KUKA KRL program: Milling_2_1.src

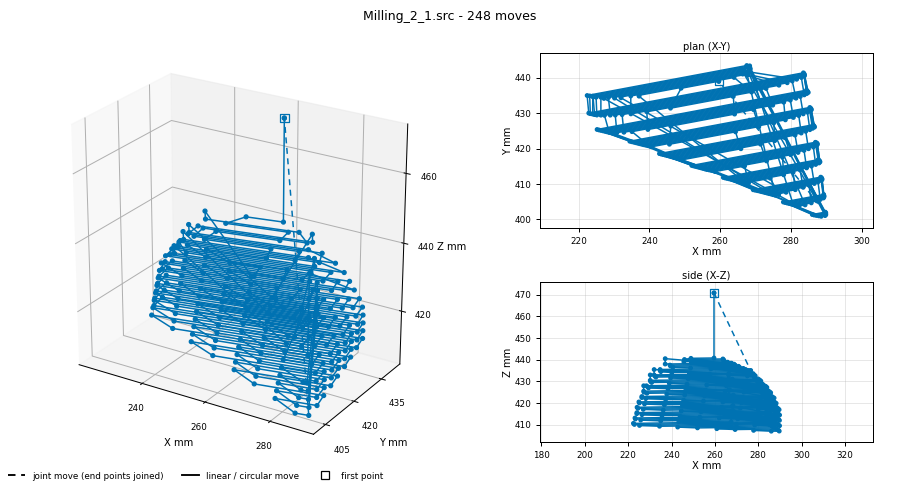
[picture p0: tool path of Milling_2_1.src, 248 of 250 moves have a stored position in this frame; points joined in program order, loops and branches not executed]
&ACCESS RVP
&REL 1
&PARAM TEMPLATE = C:\KRC\Roboter\Template\vorgabe
&PARAM EDITMASK = *
DEF Milling_2_1 ( )


;FOLD INI
;FOLD BASISTECH INI
GLOBAL INTERRUPT DECL 3 WHEN $STOPMESS==TRUE DO IR_STOPM ( )
INTERRUPT ON 3
BAS (#INITMOV,0 )
;ENDFOLD (BASISTECH INI)
;ENDFOLD (INI)

;FOLD STARTPOSITION - BASE IS 0, TOOL IS 5, SPEED IS 15%, POSITION IS A1 5,A2 -90,A3 100,A4 5,A5 -10,A6 -5,E1 0,E2 0,E3 0,E4 0
$BWDSTART = FALSE
PDAT_ACT = {VEL 15,ACC 100,APO_DIST 50}
FDAT_ACT = {TOOL_NO 5,BASE_NO 0,IPO_FRAME #BASE}
BAS (#PTP_PARAMS,15)
PTP  {A1 5,A2 -90,A3 100,A4 5,A5 -10,A6 -5,E1 0,E2 0,E3 0,E4 0}
;ENDFOLD

;FOLD LIN SPEED IS 0.1 m/sec, INTERPOLATION SETTINGS IN FOLD
$VEL.CP=0.1
$ADVANCE=3
;ENDFOLD

BAS(#VEL_PTP,2)
PTP {X 259.564, Y 439.031, Z 470.823, A 92.674, B 84.364, C 81.999, E1 0, E2 0, E3 0, E4 0, S 'B010'}
$VEL.CP=0.012
LIN {X 259.564, Y 439.031, Z 440.823, A 92.674, B 84.364, C 81.999, E1 0, E2 0, E3 0, E4 0}
LIN {X 248.928, Y 437.033, Z 440.675, A 92.674, B 84.364, C 81.999, E1 0, E2 0, E3 0, E4 0}
LIN {X 245.939, Y 431.409, Z 440.134, A 92.674, B 84.364, C 81.999, E1 0, E2 0, E3 0, E4 0}
LIN {X 263.674, Y 434.74, Z 440.381, A 92.674, B 84.364, C 81.999, E1 0, E2 0, E3 0, E4 0}
LIN {X 264.041, Y 429.745, Z 439.887, A 92.674, B 84.364, C 81.999, E1 0, E2 0, E3 0, E4 0}
LIN {X 246.004, Y 426.358, Z 439.636, A 92.674, B 84.364, C 81.999, E1 0, E2 0, E3 0, E4 0}
LIN {X 245.639, Y 421.226, Z 439.132, A 92.674, B 84.364, C 81.999, E1 0, E2 0, E3 0, E4 0}
LIN {X 264.3, Y 424.731, Z 439.392, A 92.674, B 84.364, C 81.999, E1 0, E2 0, E3 0, E4 0}
LIN {X 265.823, Y 419.953, Z 438.914, A 92.674, B 84.364, C 81.999, E1 0, E2 0, E3 0, E4 0}
LIN {X 249.117, Y 416.816, Z 438.681, A 92.674, B 84.364, C 81.999, E1 0, E2 0, E3 0, E4 0}
LIN {X 258.547, Y 413.523, Z 438.313, A 92.674, B 84.364, C 81.999, E1 0, E2 0, E3 0, E4 0}
LIN {X 266.876, Y 415.088, Z 438.429, A 92.674, B 84.364, C 81.999, E1 0, E2 0, E3 0, E4 0}
LIN {X 267.977, Y 410.231, Z 437.945, A 92.674, B 84.364, C 81.999, E1 0, E2 0, E3 0, E4 0}
LIN {X 267.316, Y 410.107, Z 437.936, A 92.674, B 84.364, C 81.999, E1 0, E2 0, E3 0, E4 0}
LIN {X 237.057, Y 434.803, Z 440.516, A 92.674, B 84.364, C 81.999, E1 0, E2 0, E3 0, E4 0}
LIN {X 237.046, Y 435.048, Z 438.028, A 92.674, B 84.364, C 81.999, E1 0, E2 0, E3 0, E4 0}
LIN {X 263.884, Y 440.089, Z 438.401, A 92.674, B 84.364, C 81.999, E1 0, E2 0, E3 0, E4 0}
LIN {X 268.845, Y 435.958, Z 437.971, A 92.674, B 84.364, C 81.999, E1 0, E2 0, E3 0, E4 0}
LIN {X 239.242, Y 430.398, Z 437.559, A 92.674, B 84.364, C 81.999, E1 0, E2 0, E3 0, E4 0}
LIN {X 239.555, Y 425.393, Z 437.064, A 92.674, B 84.364, C 81.999, E1 0, E2 0, E3 0, E4 0}
LIN {X 269.387, Y 430.996, Z 437.479, A 92.674, B 84.364, C 81.999, E1 0, E2 0, E3 0, E4 0}
LIN {X 270.891, Y 426.215, Z 437.001, A 92.674, B 84.364, C 81.999, E1 0, E2 0, E3 0, E4 0}
LIN {X 240.598, Y 420.526, Z 436.58, A 92.674, B 84.364, C 81.999, E1 0, E2 0, E3 0, E4 0}
LIN {X 248.758, Y 416.995, Z 436.194, A 92.674, B 84.364, C 81.999, E1 0, E2 0, E3 0, E4 0}
LIN {X 271.366, Y 421.241, Z 436.509, A 92.674, B 84.364, C 81.999, E1 0, E2 0, E3 0, E4 0}
LIN {X 273.07, Y 416.498, Z 436.033, A 92.674, B 84.364, C 81.999, E1 0, E2 0, E3 0, E4 0}
LIN {X 258.156, Y 413.697, Z 435.826, A 92.674, B 84.364, C 81.999, E1 0, E2 0, E3 0, E4 0}
LIN {X 266.939, Y 410.283, Z 435.449, A 92.674, B 84.364, C 81.999, E1 0, E2 0, E3 0, E4 0}
LIN {X 274.115, Y 411.631, Z 435.549, A 92.674, B 84.364, C 81.999, E1 0, E2 0, E3 0, E4 0}
LIN {X 276.51, Y 407.018, Z 435.083, A 92.674, B 84.364, C 81.999, E1 0, E2 0, E3 0, E4 0}
LIN {X 275.515, Y 406.831, Z 435.069, A 92.674, B 84.364, C 81.999, E1 0, E2 0, E3 0, E4 0}
LIN {X 267.619, Y 440.79, Z 438.464, A 92.674, B 84.364, C 81.999, E1 0, E2 0, E3 0, E4 0}
LIN {X 267.608, Y 441.035, Z 435.976, A 92.674, B 84.364, C 81.999, E1 0, E2 0, E3 0, E4 0}
LIN {X 234.715, Y 434.857, Z 435.519, A 92.674, B 84.364, C 81.999, E1 0, E2 0, E3 0, E4 0}
LIN {X 234.742, Y 429.799, Z 435.02, A 92.674, B 84.364, C 81.999, E1 0, E2 0, E3 0, E4 0}
LIN {X 272.936, Y 436.972, Z 435.551, A 92.674, B 84.364, C 81.999, E1 0, E2 0, E3 0, E4 0}
LIN {X 274.826, Y 432.264, Z 435.079, A 92.674, B 84.364, C 81.999, E1 0, E2 0, E3 0, E4 0}
LIN {X 235.05, Y 424.793, Z 434.525, A 92.674, B 84.364, C 81.999, E1 0, E2 0, E3 0, E4 0}
LIN {X 240.087, Y 420.676, Z 434.096, A 92.674, B 84.364, C 81.999, E1 0, E2 0, E3 0, E4 0}
LIN {X 275.127, Y 427.257, Z 434.584, A 92.674, B 84.364, C 81.999, E1 0, E2 0, E3 0, E4 0}
LIN {X 275.388, Y 422.243, Z 434.088, A 92.674, B 84.364, C 81.999, E1 0, E2 0, E3 0, E4 0}
LIN {X 248.208, Y 417.138, Z 433.71, A 92.674, B 84.364, C 81.999, E1 0, E2 0, E3 0, E4 0}
LIN {X 257.514, Y 413.823, Z 433.341, A 92.674, B 84.364, C 81.999, E1 0, E2 0, E3 0, E4 0}
LIN {X 277.584, Y 417.592, Z 433.62, A 92.674, B 84.364, C 81.999, E1 0, E2 0, E3 0, E4 0}
LIN {X 277.892, Y 412.587, Z 433.125, A 92.674, B 84.364, C 81.999, E1 0, E2 0, E3 0, E4 0}
LIN {X 266.359, Y 410.421, Z 432.964, A 92.674, B 84.364, C 81.999, E1 0, E2 0, E3 0, E4 0}
LIN {X 274.962, Y 406.973, Z 432.585, A 92.674, B 84.364, C 81.999, E1 0, E2 0, E3 0, E4 0}
LIN {X 278.583, Y 407.653, Z 432.635, A 92.674, B 84.364, C 81.999, E1 0, E2 0, E3 0, E4 0}
LIN {X 231.956, Y 434.337, Z 435.496, A 92.674, B 84.364, C 81.999, E1 0, E2 0, E3 0, E4 0}
LIN {X 231.944, Y 434.582, Z 433.008, A 92.674, B 84.364, C 81.999, E1 0, E2 0, E3 0, E4 0}
LIN {X 266.332, Y 441.041, Z 433.486, A 92.674, B 84.364, C 81.999, E1 0, E2 0, E3 0, E4 0}
LIN {X 276.562, Y 437.899, Z 433.129, A 92.674, B 84.364, C 81.999, E1 0, E2 0, E3 0, E4 0}
LIN {X 232.266, Y 429.58, Z 432.513, A 92.674, B 84.364, C 81.999, E1 0, E2 0, E3 0, E4 0}
LIN {X 232.779, Y 424.612, Z 432.021, A 92.674, B 84.364, C 81.999, E1 0, E2 0, E3 0, E4 0}
LIN {X 277.921, Y 433.091, Z 432.649, A 92.674, B 84.364, C 81.999, E1 0, E2 0, E3 0, E4 0}
LIN {X 278.378, Y 428.114, Z 432.156, A 92.674, B 84.364, C 81.999, E1 0, E2 0, E3 0, E4 0}
LIN {X 239.554, Y 420.822, Z 431.616, A 92.674, B 84.364, C 81.999, E1 0, E2 0, E3 0, E4 0}
LIN {X 247.69, Y 417.287, Z 431.23, A 92.674, B 84.364, C 81.999, E1 0, E2 0, E3 0, E4 0}
LIN {X 278.285, Y 423.033, Z 431.656, A 92.674, B 84.364, C 81.999, E1 0, E2 0, E3 0, E4 0}
LIN {X 279.874, Y 418.268, Z 431.179, A 92.674, B 84.364, C 81.999, E1 0, E2 0, E3 0, E4 0}
LIN {X 256.903, Y 413.954, Z 430.859, A 92.674, B 84.364, C 81.999, E1 0, E2 0, E3 0, E4 0}
LIN {X 265.846, Y 410.57, Z 430.485, A 92.674, B 84.364, C 81.999, E1 0, E2 0, E3 0, E4 0}
LIN {X 280.582, Y 413.338, Z 430.69, A 92.674, B 84.364, C 81.999, E1 0, E2 0, E3 0, E4 0}
LIN {X 281.181, Y 408.387, Z 430.199, A 92.674, B 84.364, C 81.999, E1 0, E2 0, E3 0, E4 0}
LIN {X 274.442, Y 407.121, Z 430.105, A 92.674, B 84.364, C 81.999, E1 0, E2 0, E3 0, E4 0}
LIN {X 230.149, Y 434.243, Z 433.002, A 92.674, B 84.364, C 81.999, E1 0, E2 0, E3 0, E4 0}
LIN {X 230.138, Y 434.489, Z 430.514, A 92.674, B 84.364, C 81.999, E1 0, E2 0, E3 0, E4 0}
LIN {X 266.225, Y 441.267, Z 431.016, A 92.674, B 84.364, C 81.999, E1 0, E2 0, E3 0, E4 0}
LIN {X 278.904, Y 438.585, Z 430.693, A 92.674, B 84.364, C 81.999, E1 0, E2 0, E3 0, E4 0}
LIN {X 230.334, Y 429.462, Z 430.017, A 92.674, B 84.364, C 81.999, E1 0, E2 0, E3 0, E4 0}
LIN {X 230.8, Y 424.486, Z 429.525, A 92.674, B 84.364, C 81.999, E1 0, E2 0, E3 0, E4 0}
LIN {X 279.78, Y 433.686, Z 430.206, A 92.674, B 84.364, C 81.999, E1 0, E2 0, E3 0, E4 0}
LIN {X 280.643, Y 428.785, Z 429.719, A 92.674, B 84.364, C 81.999, E1 0, E2 0, E3 0, E4 0}
LIN {X 238.939, Y 420.952, Z 429.139, A 92.674, B 84.364, C 81.999, E1 0, E2 0, E3 0, E4 0}
LIN {X 247.124, Y 417.426, Z 428.754, A 92.674, B 84.364, C 81.999, E1 0, E2 0, E3 0, E4 0}
LIN {X 281.115, Y 423.81, Z 429.226, A 92.674, B 84.364, C 81.999, E1 0, E2 0, E3 0, E4 0}
LIN {X 281.968, Y 418.907, Z 428.739, A 92.674, B 84.364, C 81.999, E1 0, E2 0, E3 0, E4 0}
LIN {X 256.243, Y 414.075, Z 428.381, A 92.674, B 84.364, C 81.999, E1 0, E2 0, E3 0, E4 0}
LIN {X 265.286, Y 410.71, Z 428.008, A 92.674, B 84.364, C 81.999, E1 0, E2 0, E3 0, E4 0}
LIN {X 282.535, Y 413.95, Z 428.248, A 92.674, B 84.364, C 81.999, E1 0, E2 0, E3 0, E4 0}
LIN {X 283.405, Y 409.05, Z 427.761, A 92.674, B 84.364, C 81.999, E1 0, E2 0, E3 0, E4 0}
LIN {X 273.873, Y 407.26, Z 427.628, A 92.674, B 84.364, C 81.999, E1 0, E2 0, E3 0, E4 0}
LIN {X 282.226, Y 403.766, Z 427.245, A 92.674, B 84.364, C 81.999, E1 0, E2 0, E3 0, E4 0}
LIN {X 283.952, Y 404.09, Z 427.269, A 92.674, B 84.364, C 81.999, E1 0, E2 0, E3 0, E4 0}
LIN {X 267.926, Y 441.584, Z 431.057, A 92.674, B 84.364, C 81.999, E1 0, E2 0, E3 0, E4 0}
LIN {X 267.915, Y 441.83, Z 428.57, A 92.674, B 84.364, C 81.999, E1 0, E2 0, E3 0, E4 0}
LIN {X 228.402, Y 434.408, Z 428.02, A 92.674, B 84.364, C 81.999, E1 0, E2 0, E3 0, E4 0}
LIN {X 228.926, Y 429.443, Z 427.528, A 92.674, B 84.364, C 81.999, E1 0, E2 0, E3 0, E4 0}
LIN {X 280.322, Y 439.097, Z 428.243, A 92.674, B 84.364, C 81.999, E1 0, E2 0, E3 0, E4 0}
LIN {X 281.379, Y 434.232, Z 427.758, A 92.674, B 84.364, C 81.999, E1 0, E2 0, E3 0, E4 0}
LIN {X 229.365, Y 424.462, Z 427.035, A 92.674, B 84.364, C 81.999, E1 0, E2 0, E3 0, E4 0}
LIN {X 238.351, Y 421.087, Z 426.661, A 92.674, B 84.364, C 81.999, E1 0, E2 0, E3 0, E4 0}
LIN {X 282.166, Y 429.316, Z 427.27, A 92.674, B 84.364, C 81.999, E1 0, E2 0, E3 0, E4 0}
LIN {X 282.861, Y 424.384, Z 426.781, A 92.674, B 84.364, C 81.999, E1 0, E2 0, E3 0, E4 0}
LIN {X 246.596, Y 417.572, Z 426.276, A 92.674, B 84.364, C 81.999, E1 0, E2 0, E3 0, E4 0}
LIN {X 255.718, Y 414.222, Z 425.904, A 92.674, B 84.364, C 81.999, E1 0, E2 0, E3 0, E4 0}
LIN {X 283.655, Y 419.469, Z 426.293, A 92.674, B 84.364, C 81.999, E1 0, E2 0, E3 0, E4 0}
LIN {X 284.384, Y 414.543, Z 425.804, A 92.674, B 84.364, C 81.999, E1 0, E2 0, E3 0, E4 0}
LIN {X 264.745, Y 410.855, Z 425.531, A 92.674, B 84.364, C 81.999, E1 0, E2 0, E3 0, E4 0}
LIN {X 273.326, Y 407.403, Z 425.151, A 92.674, B 84.364, C 81.999, E1 0, E2 0, E3 0, E4 0}
LIN {X 285.08, Y 409.61, Z 425.314, A 92.674, B 84.364, C 81.999, E1 0, E2 0, E3 0, E4 0}
LIN {X 285.706, Y 404.665, Z 424.824, A 92.674, B 84.364, C 81.999, E1 0, E2 0, E3 0, E4 0}
LIN {X 281.681, Y 403.909, Z 424.768, A 92.674, B 84.364, C 81.999, E1 0, E2 0, E3 0, E4 0}
LIN {X 227.131, Y 434.168, Z 428.021, A 92.674, B 84.364, C 81.999, E1 0, E2 0, E3 0, E4 0}
LIN {X 227.12, Y 434.413, Z 425.533, A 92.674, B 84.364, C 81.999, E1 0, E2 0, E3 0, E4 0}
LIN {X 266.806, Y 441.867, Z 426.085, A 92.674, B 84.364, C 81.999, E1 0, E2 0, E3 0, E4 0}
LIN {X 281.564, Y 439.576, Z 425.791, A 92.674, B 84.364, C 81.999, E1 0, E2 0, E3 0, E4 0}
LIN {X 227.291, Y 429.382, Z 425.036, A 92.674, B 84.364, C 81.999, E1 0, E2 0, E3 0, E4 0}
LIN {X 228.634, Y 424.571, Z 424.556, A 92.674, B 84.364, C 81.999, E1 0, E2 0, E3 0, E4 0}
LIN {X 282.602, Y 434.707, Z 425.307, A 92.674, B 84.364, C 81.999, E1 0, E2 0, E3 0, E4 0}
LIN {X 283.429, Y 429.799, Z 424.819, A 92.674, B 84.364, C 81.999, E1 0, E2 0, E3 0, E4 0}
LIN {X 237.795, Y 421.228, Z 424.184, A 92.674, B 84.364, C 81.999, E1 0, E2 0, E3 0, E4 0}
LIN {X 246.074, Y 417.72, Z 423.8, A 92.674, B 84.364, C 81.999, E1 0, E2 0, E3 0, E4 0}
LIN {X 284.128, Y 424.867, Z 424.33, A 92.674, B 84.364, C 81.999, E1 0, E2 0, E3 0, E4 0}
LIN {X 284.909, Y 419.951, Z 423.842, A 92.674, B 84.364, C 81.999, E1 0, E2 0, E3 0, E4 0}
LIN {X 255.198, Y 414.37, Z 423.428, A 92.674, B 84.364, C 81.999, E1 0, E2 0, E3 0, E4 0}
LIN {X 264.209, Y 410.999, Z 423.054, A 92.674, B 84.364, C 81.999, E1 0, E2 0, E3 0, E4 0}
LIN {X 285.756, Y 415.046, Z 423.354, A 92.674, B 84.364, C 81.999, E1 0, E2 0, E3 0, E4 0}
LIN {X 286.552, Y 410.133, Z 422.866, A 92.674, B 84.364, C 81.999, E1 0, E2 0, E3 0, E4 0}
LIN {X 272.782, Y 407.546, Z 422.675, A 92.674, B 84.364, C 81.999, E1 0, E2 0, E3 0, E4 0}
LIN {X 281.14, Y 404.053, Z 422.292, A 92.674, B 84.364, C 81.999, E1 0, E2 0, E3 0, E4 0}
LIN {X 287.285, Y 405.207, Z 422.377, A 92.674, B 84.364, C 81.999, E1 0, E2 0, E3 0, E4 0}
LIN {X 266.32, Y 441.774, Z 426.097, A 92.674, B 84.364, C 81.999, E1 0, E2 0, E3 0, E4 0}
LIN {X 266.309, Y 442.019, Z 423.609, A 92.674, B 84.364, C 81.999, E1 0, E2 0, E3 0, E4 0}
LIN {X 226.275, Y 434.5, Z 423.053, A 92.674, B 84.364, C 81.999, E1 0, E2 0, E3 0, E4 0}
LIN {X 226.277, Y 429.437, Z 422.554, A 92.674, B 84.364, C 81.999, E1 0, E2 0, E3 0, E4 0}
LIN {X 282.895, Y 440.071, Z 423.341, A 92.674, B 84.364, C 81.999, E1 0, E2 0, E3 0, E4 0}
LIN {X 283.716, Y 435.162, Z 422.853, A 92.674, B 84.364, C 81.999, E1 0, E2 0, E3 0, E4 0}
LIN {X 228.078, Y 424.712, Z 422.079, A 92.674, B 84.364, C 81.999, E1 0, E2 0, E3 0, E4 0}
LIN {X 237.249, Y 421.371, Z 421.708, A 92.674, B 84.364, C 81.999, E1 0, E2 0, E3 0, E4 0}
LIN {X 284.613, Y 430.267, Z 422.367, A 92.674, B 84.364, C 81.999, E1 0, E2 0, E3 0, E4 0}
LIN {X 285.293, Y 425.332, Z 421.877, A 92.674, B 84.364, C 81.999, E1 0, E2 0, E3 0, E4 0}
LIN {X 245.557, Y 417.868, Z 421.324, A 92.674, B 84.364, C 81.999, E1 0, E2 0, E3 0, E4 0}
LIN {X 254.682, Y 414.519, Z 420.952, A 92.674, B 84.364, C 81.999, E1 0, E2 0, E3 0, E4 0}
LIN {X 286.287, Y 420.455, Z 421.392, A 92.674, B 84.364, C 81.999, E1 0, E2 0, E3 0, E4 0}
LIN {X 286.935, Y 415.513, Z 420.902, A 92.674, B 84.364, C 81.999, E1 0, E2 0, E3 0, E4 0}
LIN {X 263.676, Y 411.145, Z 420.578, A 92.674, B 84.364, C 81.999, E1 0, E2 0, E3 0, E4 0}
LIN {X 272.241, Y 407.69, Z 420.198, A 92.674, B 84.364, C 81.999, E1 0, E2 0, E3 0, E4 0}
LIN {X 287.6, Y 410.575, Z 420.412, A 92.674, B 84.364, C 81.999, E1 0, E2 0, E3 0, E4 0}
LIN {X 288.242, Y 405.632, Z 419.922, A 92.674, B 84.364, C 81.999, E1 0, E2 0, E3 0, E4 0}
LIN {X 280.602, Y 404.197, Z 419.815, A 92.674, B 84.364, C 81.999, E1 0, E2 0, E3 0, E4 0}
LIN {X 268.441, Y 442.417, Z 423.66, A 92.674, B 84.364, C 81.999, E1 0, E2 0, E3 0, E4 0}
LIN {X 268.429, Y 442.663, Z 421.172, A 92.674, B 84.364, C 81.999, E1 0, E2 0, E3 0, E4 0}
LIN {X 224.921, Y 434.491, Z 420.567, A 92.674, B 84.364, C 81.999, E1 0, E2 0, E3 0, E4 0}
LIN {X 225.137, Y 429.468, Z 420.071, A 92.674, B 84.364, C 81.999, E1 0, E2 0, E3 0, E4 0}
LIN {X 283.71, Y 440.469, Z 420.885, A 92.674, B 84.364, C 81.999, E1 0, E2 0, E3 0, E4 0}
LIN {X 284.438, Y 435.543, Z 420.396, A 92.674, B 84.364, C 81.999, E1 0, E2 0, E3 0, E4 0}
LIN {X 227.507, Y 424.85, Z 419.604, A 92.674, B 84.364, C 81.999, E1 0, E2 0, E3 0, E4 0}
LIN {X 236.686, Y 421.511, Z 419.233, A 92.674, B 84.364, C 81.999, E1 0, E2 0, E3 0, E4 0}
LIN {X 285.251, Y 430.632, Z 419.909, A 92.674, B 84.364, C 81.999, E1 0, E2 0, E3 0, E4 0}
LIN {X 286.064, Y 425.722, Z 419.421, A 92.674, B 84.364, C 81.999, E1 0, E2 0, E3 0, E4 0}
LIN {X 245.014, Y 418.011, Z 418.85, A 92.674, B 84.364, C 81.999, E1 0, E2 0, E3 0, E4 0}
LIN {X 254.14, Y 414.662, Z 418.477, A 92.674, B 84.364, C 81.999, E1 0, E2 0, E3 0, E4 0}
LIN {X 287.126, Y 420.858, Z 418.936, A 92.674, B 84.364, C 81.999, E1 0, E2 0, E3 0, E4 0}
LIN {X 287.884, Y 415.937, Z 418.448, A 92.674, B 84.364, C 81.999, E1 0, E2 0, E3 0, E4 0}
LIN {X 263.134, Y 411.288, Z 418.103, A 92.674, B 84.364, C 81.999, E1 0, E2 0, E3 0, E4 0}
LIN {X 271.675, Y 407.829, Z 417.723, A 92.674, B 84.364, C 81.999, E1 0, E2 0, E3 0, E4 0}
LIN {X 288.527, Y 410.994, Z 417.957, A 92.674, B 84.364, C 81.999, E1 0, E2 0, E3 0, E4 0}
LIN {X 289.124, Y 406.043, Z 417.467, A 92.674, B 84.364, C 81.999, E1 0, E2 0, E3 0, E4 0}
LIN {X 280.035, Y 404.336, Z 417.34, A 92.674, B 84.364, C 81.999, E1 0, E2 0, E3 0, E4 0}
LIN {X 288.51, Y 400.865, Z 416.959, A 92.674, B 84.364, C 81.999, E1 0, E2 0, E3 0, E4 0}
LIN {X 289.6, Y 401.069, Z 416.974, A 92.674, B 84.364, C 81.999, E1 0, E2 0, E3 0, E4 0}
LIN {X 268.254, Y 442.628, Z 421.191, A 92.674, B 84.364, C 81.999, E1 0, E2 0, E3 0, E4 0}
LIN {X 268.243, Y 442.873, Z 418.703, A 92.674, B 84.364, C 81.999, E1 0, E2 0, E3 0, E4 0}
LIN {X 224.071, Y 434.576, Z 418.088, A 92.674, B 84.364, C 81.999, E1 0, E2 0, E3 0, E4 0}
LIN {X 224.497, Y 429.593, Z 417.595, A 92.674, B 84.364, C 81.999, E1 0, E2 0, E3 0, E4 0}
LIN {X 283.792, Y 440.73, Z 418.42, A 92.674, B 84.364, C 81.999, E1 0, E2 0, E3 0, E4 0}
LIN {X 284.855, Y 435.867, Z 417.935, A 92.674, B 84.364, C 81.999, E1 0, E2 0, E3 0, E4 0}
LIN {X 226.935, Y 424.988, Z 417.13, A 92.674, B 84.364, C 81.999, E1 0, E2 0, E3 0, E4 0}
LIN {X 236.143, Y 421.654, Z 416.759, A 92.674, B 84.364, C 81.999, E1 0, E2 0, E3 0, E4 0}
LIN {X 285.726, Y 430.967, Z 417.448, A 92.674, B 84.364, C 81.999, E1 0, E2 0, E3 0, E4 0}
LIN {X 286.616, Y 426.071, Z 416.962, A 92.674, B 84.364, C 81.999, E1 0, E2 0, E3 0, E4 0}
LIN {X 244.47, Y 418.155, Z 416.375, A 92.674, B 84.364, C 81.999, E1 0, E2 0, E3 0, E4 0}
LIN {X 253.598, Y 414.806, Z 416.003, A 92.674, B 84.364, C 81.999, E1 0, E2 0, E3 0, E4 0}
LIN {X 287.417, Y 421.158, Z 416.474, A 92.674, B 84.364, C 81.999, E1 0, E2 0, E3 0, E4 0}
LIN {X 288.158, Y 416.234, Z 415.985, A 92.674, B 84.364, C 81.999, E1 0, E2 0, E3 0, E4 0}
LIN {X 262.569, Y 411.428, Z 415.629, A 92.674, B 84.364, C 81.999, E1 0, E2 0, E3 0, E4 0}
LIN {X 271.128, Y 407.972, Z 415.249, A 92.674, B 84.364, C 81.999, E1 0, E2 0, E3 0, E4 0}
LIN {X 288.749, Y 411.281, Z 415.494, A 92.674, B 84.364, C 81.999, E1 0, E2 0, E3 0, E4 0}
LIN {X 289.25, Y 406.312, Z 415.002, A 92.674, B 84.364, C 81.999, E1 0, E2 0, E3 0, E4 0}
LIN {X 279.481, Y 404.477, Z 414.866, A 92.674, B 84.364, C 81.999, E1 0, E2 0, E3 0, E4 0}
LIN {X 287.851, Y 400.986, Z 414.483, A 92.674, B 84.364, C 81.999, E1 0, E2 0, E3 0, E4 0}
LIN {X 289.817, Y 401.355, Z 414.511, A 92.674, B 84.364, C 81.999, E1 0, E2 0, E3 0, E4 0}
LIN {X 268.187, Y 442.86, Z 418.725, A 92.674, B 84.364, C 81.999, E1 0, E2 0, E3 0, E4 0}
LIN {X 268.176, Y 443.105, Z 416.237, A 92.674, B 84.364, C 81.999, E1 0, E2 0, E3 0, E4 0}
LIN {X 224.001, Y 434.808, Z 415.623, A 92.674, B 84.364, C 81.999, E1 0, E2 0, E3 0, E4 0}
LIN {X 223.955, Y 429.736, Z 415.123, A 92.674, B 84.364, C 81.999, E1 0, E2 0, E3 0, E4 0}
LIN {X 283.74, Y 440.966, Z 415.954, A 92.674, B 84.364, C 81.999, E1 0, E2 0, E3 0, E4 0}
LIN {X 284.674, Y 436.078, Z 415.468, A 92.674, B 84.364, C 81.999, E1 0, E2 0, E3 0, E4 0}
LIN {X 226.342, Y 425.121, Z 414.657, A 92.674, B 84.364, C 81.999, E1 0, E2 0, E3 0, E4 0}
LIN {X 235.578, Y 421.793, Z 414.286, A 92.674, B 84.364, C 81.999, E1 0, E2 0, E3 0, E4 0}
LIN {X 285.654, Y 431.198, Z 414.983, A 92.674, B 84.364, C 81.999, E1 0, E2 0, E3 0, E4 0}
LIN {X 286.529, Y 426.299, Z 414.496, A 92.674, B 84.364, C 81.999, E1 0, E2 0, E3 0, E4 0}
LIN {X 243.906, Y 418.294, Z 413.903, A 92.674, B 84.364, C 81.999, E1 0, E2 0, E3 0, E4 0}
LIN {X 253.035, Y 414.945, Z 413.531, A 92.674, B 84.364, C 81.999, E1 0, E2 0, E3 0, E4 0}
LIN {X 287.404, Y 421.4, Z 414.009, A 92.674, B 84.364, C 81.999, E1 0, E2 0, E3 0, E4 0}
LIN {X 288.081, Y 416.464, Z 413.519, A 92.674, B 84.364, C 81.999, E1 0, E2 0, E3 0, E4 0}
LIN {X 261.964, Y 411.559, Z 413.156, A 92.674, B 84.364, C 81.999, E1 0, E2 0, E3 0, E4 0}
LIN {X 270.536, Y 408.106, Z 412.776, A 92.674, B 84.364, C 81.999, E1 0, E2 0, E3 0, E4 0}
LIN {X 288.692, Y 411.516, Z 413.029, A 92.674, B 84.364, C 81.999, E1 0, E2 0, E3 0, E4 0}
LIN {X 289.326, Y 406.572, Z 412.538, A 92.674, B 84.364, C 81.999, E1 0, E2 0, E3 0, E4 0}
LIN {X 278.912, Y 404.615, Z 412.393, A 92.674, B 84.364, C 81.999, E1 0, E2 0, E3 0, E4 0}
LIN {X 287.17, Y 401.103, Z 412.009, A 92.674, B 84.364, C 81.999, E1 0, E2 0, E3 0, E4 0}
LIN {X 289.754, Y 401.589, Z 412.045, A 92.674, B 84.364, C 81.999, E1 0, E2 0, E3 0, E4 0}
LIN {X 268.312, Y 443.129, Z 416.261, A 92.674, B 84.364, C 81.999, E1 0, E2 0, E3 0, E4 0}
LIN {X 268.301, Y 443.374, Z 413.773, A 92.674, B 84.364, C 81.999, E1 0, E2 0, E3 0, E4 0}
LIN {X 223.107, Y 434.886, Z 413.145, A 92.674, B 84.364, C 81.999, E1 0, E2 0, E3 0, E4 0}
LIN {X 223.296, Y 429.858, Z 412.648, A 92.674, B 84.364, C 81.999, E1 0, E2 0, E3 0, E4 0}
LIN {X 283.609, Y 441.186, Z 413.487, A 92.674, B 84.364, C 81.999, E1 0, E2 0, E3 0, E4 0}
LIN {X 284.539, Y 436.298, Z 413.001, A 92.674, B 84.364, C 81.999, E1 0, E2 0, E3 0, E4 0}
LIN {X 225.754, Y 425.256, Z 412.183, A 92.674, B 84.364, C 81.999, E1 0, E2 0, E3 0, E4 0}
LIN {X 235.006, Y 421.931, Z 411.813, A 92.674, B 84.364, C 81.999, E1 0, E2 0, E3 0, E4 0}
LIN {X 285.501, Y 431.415, Z 412.515, A 92.674, B 84.364, C 81.999, E1 0, E2 0, E3 0, E4 0}
LIN {X 286.303, Y 426.502, Z 412.027, A 92.674, B 84.364, C 81.999, E1 0, E2 0, E3 0, E4 0}
LIN {X 243.349, Y 418.434, Z 411.43, A 92.674, B 84.364, C 81.999, E1 0, E2 0, E3 0, E4 0}
LIN {X 252.481, Y 415.086, Z 411.058, A 92.674, B 84.364, C 81.999, E1 0, E2 0, E3 0, E4 0}
LIN {X 287.204, Y 421.608, Z 411.541, A 92.674, B 84.364, C 81.999, E1 0, E2 0, E3 0, E4 0}
LIN {X 287.881, Y 416.672, Z 411.051, A 92.674, B 84.364, C 81.999, E1 0, E2 0, E3 0, E4 0}
LIN {X 261.392, Y 411.697, Z 410.683, A 92.674, B 84.364, C 81.999, E1 0, E2 0, E3 0, E4 0}
LIN {X 269.901, Y 408.232, Z 410.302, A 92.674, B 84.364, C 81.999, E1 0, E2 0, E3 0, E4 0}
LIN {X 288.582, Y 411.74, Z 410.562, A 92.674, B 84.364, C 81.999, E1 0, E2 0, E3 0, E4 0}
LIN {X 289.202, Y 406.793, Z 410.071, A 92.674, B 84.364, C 81.999, E1 0, E2 0, E3 0, E4 0}
LIN {X 278.351, Y 404.755, Z 409.92, A 92.674, B 84.364, C 81.999, E1 0, E2 0, E3 0, E4 0}
LIN {X 286.517, Y 401.226, Z 409.535, A 92.674, B 84.364, C 81.999, E1 0, E2 0, E3 0, E4 0}
LIN {X 289.801, Y 401.843, Z 409.58, A 92.674, B 84.364, C 81.999, E1 0, E2 0, E3 0, E4 0}
LIN {X 267.483, Y 443.219, Z 413.783, A 92.674, B 84.364, C 81.999, E1 0, E2 0, E3 0, E4 0}
LIN {X 267.472, Y 443.464, Z 411.295, A 92.674, B 84.364, C 81.999, E1 0, E2 0, E3 0, E4 0}
LIN {X 222.393, Y 434.997, Z 410.668, A 92.674, B 84.364, C 81.999, E1 0, E2 0, E3 0, E4 0}
LIN {X 222.85, Y 430.02, Z 410.175, A 92.674, B 84.364, C 81.999, E1 0, E2 0, E3 0, E4 0}
LIN {X 283.471, Y 441.406, Z 411.018, A 92.674, B 84.364, C 81.999, E1 0, E2 0, E3 0, E4 0}
LIN {X 284.338, Y 436.505, Z 410.531, A 92.674, B 84.364, C 81.999, E1 0, E2 0, E3 0, E4 0}
LIN {X 225.2, Y 425.397, Z 409.708, A 92.674, B 84.364, C 81.999, E1 0, E2 0, E3 0, E4 0}
LIN {X 234.441, Y 422.07, Z 409.338, A 92.674, B 84.364, C 81.999, E1 0, E2 0, E3 0, E4 0}
LIN {X 285.282, Y 431.619, Z 410.045, A 92.674, B 84.364, C 81.999, E1 0, E2 0, E3 0, E4 0}
LIN {X 286.186, Y 426.725, Z 409.559, A 92.674, B 84.364, C 81.999, E1 0, E2 0, E3 0, E4 0}
LIN {X 242.819, Y 418.58, Z 408.955, A 92.674, B 84.364, C 81.999, E1 0, E2 0, E3 0, E4 0}
LIN {X 251.949, Y 415.232, Z 408.583, A 92.674, B 84.364, C 81.999, E1 0, E2 0, E3 0, E4 0}
LIN {X 286.863, Y 421.789, Z 409.069, A 92.674, B 84.364, C 81.999, E1 0, E2 0, E3 0, E4 0}
LIN {X 287.627, Y 416.869, Z 408.58, A 92.674, B 84.364, C 81.999, E1 0, E2 0, E3 0, E4 0}
LIN {X 260.857, Y 411.841, Z 408.208, A 92.674, B 84.364, C 81.999, E1 0, E2 0, E3 0, E4 0}
LIN {X 269.303, Y 408.365, Z 407.826, A 92.674, B 84.364, C 81.999, E1 0, E2 0, E3 0, E4 0}
LIN {X 288.361, Y 411.944, Z 408.091, A 92.674, B 84.364, C 81.999, E1 0, E2 0, E3 0, E4 0}
LIN {X 289.206, Y 407.039, Z 407.604, A 92.674, B 84.364, C 81.999, E1 0, E2 0, E3 0, E4 0}
LIN {X 277.82, Y 404.901, Z 407.446, A 92.674, B 84.364, C 81.999, E1 0, E2 0, E3 0, E4 0}
LIN {X 285.985, Y 401.371, Z 407.06, A 92.674, B 84.364, C 81.999, E1 0, E2 0, E3 0, E4 0}
LIN {X 289.657, Y 402.061, Z 407.111, A 92.674, B 84.364, C 81.999, E1 0, E2 0, E3 0, E4 0}
PTP {X 259.564, Y 439.031, Z 470.823, A 92.674, B 84.364, C 81.999, E1 0, E2 0, E3 0, E4 0, S 'B010'}
PTP {A1 5, A2 -90, A3 100, A4 5, A5 -10, A6 -5, E1 0, E2 0, E3 0, E4 0} C_PTP

END
